FUNCTION acc_dec : bool
VAR_INPUT
	a	:	BOOL;
	d	:	BOOL;
END_VAR
VAR
END_VAR

//	setting coeficient state 
generalVariable.staus.Accel := a;
generalVariable.staus.Decel := d;

END_FUNCTION

(* stored: Version 1.1.0.1, ProductVersion 3.1.4024.12
   POU acc_dec: Id {a5b21f10-7429-450c-88b6-f83d69bc1575}, SpecialFunc None *)
